FUNCTION_BLOCK HAL_DO_Channel IMPLEMENTS I_HAL_DO
VAR_INPUT
	terminal_address		: WORD;
END_VAR
VAR_OUTPUT
END_VAR
VAR
	_terminal_value: BOOL;
	_errId:HAL_ErrorEnum;
	_xValue: BOOL;
	_channel_number: UINT;
END_VAR

PROPERTY errId : HAL_ErrorEnum
GET
errId := _errId;
END_GET
END_PROPERTY

METHOD FB_init : BOOL
VAR_INPUT
	bInitRetains 	: BOOL; // if TRUE, the retain variables are initialized (warm start / cold start)
	bInCopyCode 	: BOOL;  // if TRUE, the instance afterwards gets moved into the copy code (online change)
    channel_number  : UINT;
END_VAR

_channel_number :=channel_number;
END_METHOD

PROPERTY terminal_value : bool
GET
terminal_value := _xValue;
END_GET
END_PROPERTY

PROPERTY WcState : bool
GET
END_GET
SET
END_SET
END_PROPERTY

PROPERTY xValue : BOOL
GET
xValue:=_xValue;
END_GET
SET
_xValue := xValue;
END_SET
END_PROPERTY

END_FUNCTION_BLOCK

(* stored: Version 1.1.0.1, ProductVersion 3.1.4024.6
   POU HAL_DO_Channel: Id {4b567117-22ec-0e75-3dff-6e4001d998ad}, SpecialFunc None
   Folder HAL: Id {4d92782d-af7a-0573-1cd5-f1b8218525dd}
   Folder IO: Id {5c56663d-53d8-0172-3815-e08520cf184c}
   Property errId: Id {7c6bdd6e-b6f5-06fb-2802-0ffb22035f06}
   Get Get: Id {12faf0f8-1c53-0a55-3856-3e132c58eb46}
   Method FB_init: Id {2e7e34e1-a708-0df8-265e-0041b8f882e4}
   Property terminal_value: Id {7eaf041c-d0a1-0190-1dac-dcd942191d21}
   Get Get: Id {eb382bbf-9081-026a-1776-50932c766bf9}
   Property WcState: Id {b71a6f61-ff21-0e16-3e20-04d7b17415d0}
   Get Get: Id {6905b1cf-74d1-0984-317f-aba3bf7ec6b9}
   Set Set: Id {25c4b58b-1328-0246-1def-c1c762232b24}
   Property xValue: Id {6dddd416-6bcf-07da-2740-e7b561c5554d}
   Get Get: Id {b777ab7b-d03e-0284-1db8-8eee7fbd572b}
   Set Set: Id {329a4166-b2f0-0187-3fcd-586230b79595} *)
